TYPE TcoUrRobotics_T2O_BitRegs_IO :
STRUCT
    bArray AT %I* : ARRAY[0..7] OF BYTE;
END_STRUCT
END_TYPE

(* stored: Version 1.1.0.1, ProductVersion 3.1.4024.12
   DUT TcoUrRobotics_T2O_BitRegs_IO: Id {1df4fb15-c339-0f7b-1cbc-c02b1c445054} *)
